TYPE TcaCarrierService :
STRUCT

END_STRUCT
END_TYPE

(* stored: Version 1.1.0.1
   DUT TcaCarrierService: Id {a05e7cbc-b3a7-482a-a741-a868c9d381ac} *)
